FUNCTION_BLOCK CU030ManualTask EXTENDS TcoTaskedService IMPLEMENTS ICUTask
VAR
END_VAR

Run();

(*~
	<docu>
		<summary>
			Main method of the sequener. Custom code needs to be placed here. The sequencer is executed by call of **Instance.Run()** method.
			This method is abstract, and it must be overridden in derived block.
		</summary>
	</docu>
~*)
METHOD PROTECTED Main : BOOL
Messenger.Notify('Running manual mode');
Station.Components.Group1.horizontalCylinder.Service();
END_METHOD

METHOD PROTECTED OnStart
Station.AutomatTask.Restore();
Station.GroundTask.Restore();
Station.GroundTask.CancelGround();
END_METHOD

PROPERTY Station : REFERENCE TO CU030
GET
VAR
    _station : POINTER TO CU030;
END_VAR
IF __QUERYPOINTER(Parent, _station) THEN // Check if _Parent is Station001
    Station REF= _station^;              // If the check is successful dereference a pointer. simlar to THIS^ or SUPER^
END_IF
END_GET
END_PROPERTY

END_FUNCTION_BLOCK

(* stored: Version 1.1.0.1
   POU CU030ManualTask: Id {2b7d0710-c2fb-4ff0-b058-7caf4008048d}, SpecialFunc None
   Method Main: Id {64a43192-21c8-4e89-b80f-3be0695c8348}
   Method OnStart: Id {946b540d-738b-43a1-a72d-e2687f7b530a}
   Property Station: Id {5259f7e6-2875-406b-9435-da43004c0e1a}
   Get Get: Id {2b862502-e2f1-4cca-af35-78c4cd405706} *)
